// TIA Portal V18 export
DATA_BLOCK "SpeedAxis_1"   // DB2, Motion_DB
// stored: AutoNumber true, DBAccessibleFromOPCUA true, DBAccessibleFromWebserver true, InstanceOfName TO_SpeedAxis, OfSystemLibElement TO_SpeedAxis, OfSystemLibVersion 7.0
TO_SpeedAxis   // technology object, version 7.0
// stored: Connection Interface Actor
// stored: Connection Interface Torque
   // // inherited from TO_Axis
   // // inherited from TO_Object
   // VAR
   //    Velocity { ExternalWritable := 'False'} : LReal;
   //    Acceleration { ExternalWritable := 'False'} : LReal;
   //    ActualSpeed { ExternalWritable := 'False'} : LReal;
   //    VelocitySetpoint { ExternalWritable := 'False'} : LReal;
   //    Actor { S7_SetPoint := 'True'} : TO_Struct_Actor;
   //    TorqueLimiting { S7_SetPoint := 'True'} : TO_Struct_TorqueLimiting;
   //    LoadGear { S7_SetPoint := 'True'} : TO_Struct_LoadGear;
   //    DynamicLimits { S7_SetPoint := 'True'} : TO_Struct_DynamicLimits;
   //    DynamicDefaults { S7_SetPoint := 'True'} : TO_Struct_DynamicDefaults;
   //    Override { S7_SetPoint := 'True'} : TO_Struct_Override;
   //    Units { ExternalWritable := 'False'; S7_SetPoint := 'True'} : TO_Struct_Units;
   //    StatusDrive { ExternalWritable := 'False'; S7_SetPoint := 'True'} : TO_Struct_StatusDrive;
   //    StatusTorqueData { ExternalWritable := 'False'; S7_SetPoint := 'True'} : TO_Struct_StatusTorqueData;
   //    StatusMotionIn { ExternalWritable := 'False'; S7_SetPoint := 'True'} : TO_Struct_StatusMotionIn;
   //    StatusWord { ExternalWritable := 'False'} : DWord;
   //    StatusWord2 { ExternalWritable := 'False'} : DWord;
   //    ErrorWord { ExternalWritable := 'False'} : DWord;
   //    ErrorDetail { ExternalWritable := 'False'; S7_SetPoint := 'True'} : TO_Struct_ErrorDetail;
   //    WarningWord { ExternalWritable := 'False'} : DWord;
   //    ControlPanel { S7_SetPoint := 'True'} : TO_Struct_ControlPanel;
   //    InternalToTrace { S7_SetPoint := 'True'} : Array[1..4] of TO_Struct_Internal;
   //    VirtualAxis { ExternalWritable := 'False'; S7_SetPoint := 'True'} : TO_Struct_VirtualAxis;
   //    Simulation { S7_SetPoint := 'True'} : TO_Struct_AxisSimulation;
   // END_VAR
BEGIN
   DynamicLimits.MaxAcceleration := 1000.0;
   DynamicLimits.MaxDeceleration := 1000.0;
   DynamicLimits.MaxJerk := 20000.0;
   DynamicDefaults.Acceleration := 200.0;
   DynamicDefaults.Deceleration := 200.0;
   DynamicDefaults.Jerk := 4000.0;
   DynamicDefaults.EmergencyDeceleration := 1000.0;
   VirtualAxis.Mode := 1;
   VirtualAxis.Mode := 1;
END_DATA_BLOCK
